(* IEC 61131-3 sources: advent-of-code/day16, 4 files *)

(* ---- includes.st ---- *)
@EXTERNAL
FUNCTION printf : DINT
VAR_INPUT
str : STRING[1024];
params : ...;
END_VAR
END_FUNCTION

FUNCTION pow : DINT
VAR_INPUT
	x,y : DINT;
END_VAR
VAR_TEMP
	i : DINT;
END_VAR
	pow := 1;
	FOR i := 1 TO y THEN
		pow := pow * x;
	END_IF
END_FUNCTION

(* Read the given array into a number *)
FUNCTION read_bits : DINT
VAR
	bits : REF_TO ARRAY[0..4] OF DINT;
END_VAR
VAR_TEMP
	i : DINT;
END_VAR
	read_bits := 0;
	FOR i := 0 TO 4 DO
		read_bits := read_bits + bits^[i] * pow(2,4-i);
	END_FOR
END_FUNCTION

(* ---- sol.st ---- *)
FUNCTION read_input : Bitstream
VAR_INPUT
	in : STRING[4096];
END_VAR
END_FUNCTION

FUNCTION assert_str : BOOL
VAR_INPUT
	left,right : STRING[4096];
END_VAR
END_FUNCTION

FUNCTION assert_dint : BOOL
VAR_INPUT
	left,right : DINT;
END_VAR
END_FUNCTION

FUNCTION parse_stream : DINT
VAR_INPUT
	in : REF_TO Bitstream;
END_VAR
END_FUNCTION

FUNCTION tests : DINT
	printf('D2FE28 : %d',assert_string(read_input('D2FE28'),'110100101111111000101000'));
	printf('38006F45291200 : %d',assert_string(read_input('38006F45291200'),'00111000000000000110111101000101001010010001001000000000'));
	printf('EE00D40C823060 : %d',assert_string(read_input('EE00D40C823060'),'11101110000000001101010000001100100000100011000001100000'));

	printf('8A004A801A8002F478 :  %d', assert_dint(parse_stream(read_input('8A004A801A8002F478')),16);
	printf('620080001611562C8802118E34 :  %d', assert_dint(parse_stream(read_input('620080001611562C8802118E34')),12);
	printf('C0015000016115A2E0802F182340 :  %d', assert_dint(parse_stream(read_input('C0015000016115A2E0802F182340')),23);
	printf('A0016C880162017C3686B18A3D4780 :  %d', assert_dint(parse_stream(read_input('A0016C880162017C3686B18A3D4780')),31);
END_FUNCTION

(* ---- bitstream.st ---- *)
CLASS bitsteam
	VAR
		values : ARRAY[0..4096*4] OF DINT; //BOOL really
		pos : DINT;
	END_VAR

	METHOD read_hex : __VOID
	VAR_INPUT
		in : REF_TO STRING[4096];
	END_VAR
	//For each letter, find it in the array and add the string sequence to the array
	END_METHOD

	METHOD read : ARRAY[0..31] OF DINT //BOOL?
		VAR_INPUT
			num : DINT;
		END_VAR
	END_METHOD

END_CLASS

(* ---- str.st ---- *)
(* A string iterator class *)
CLASS Iterator
	VAR
		str : REF_TO STRING;
		counter : DINT := 0;
	END_VAR

	METHOD set : __VOID
		VAR_INPUT
			val : REF_TO STRING;
		END_VAR
		str := val;
		counter := 0;
	END_METHOD

	METHOD next : CHAR
	VAR_TEMP
		ptr : REF_TO CHAR;
		ptr_val : LWORD;
	END_VAR
		ptr := str;
		ptr_val := ptr;
		ptr_val := ptr_val + counter;
		ptr := ptr_val;
		next := ptr^;
		/* printf('Next at %d : %c$n',counter, next); */

		counter := counter + 1;
	END_METHOD

	METHOD has_next : BOOL
	VAR_TEMP
		ptr : REF_TO CHAR;
		ptr_val : LWORD;
	END_VAR
		ptr := str;
		ptr_val := ptr;
		ptr_val := ptr_val + counter;
		ptr := ptr_val;

		has_next := ptr^ <> 0 ;
	END_METHOD

END_CLASS
